FUNCTION_BLOCK SPINNER (* Spinner for UINT{0..100} input *)
  (* Standard: 61499-1; Classification: HMI *)
  (* Version 0.1, 2007-09-03, JHC, Holobloc Inc *)
  (* Version 0.0, 2007-08-30, JHC, Holobloc Inc *)
  (* Compiler header: package fb.rt.hmi; *)
  (* Compiler Java Sun JDK 1.6.0 *)
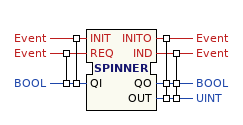
  EVENT_INPUT
    INIT WITH QI; (* Initialization *)
    REQ WITH QI; (* Request *)
  END_EVENT
  EVENT_OUTPUT
    INITO WITH QO, OUT; (* Initialization Confirm *)
    IND WITH QO, OUT; (* User changed choice or REQ serviced *)
  END_EVENT
  VAR_INPUT
    QI : BOOL := true; (* Input Event Qualifier / Output Enable *)
  END_VAR
  VAR_OUTPUT
    QO : BOOL; (* Event Qualifier *)
    OUT : UINT; (* Current Spinner Value {0..100} *)
  END_VAR
END_FUNCTION_BLOCK
